FUNCTION_BLOCK PalletizerConveyor EXTENDS Conveyor
VAR_INPUT
END_VAR
VAR_OUTPUT
	bStartBackward : BOOL;
END_VAR
VAR	
	fbStartBackward : BoolOut;
END_VAR

SUPER^();
bStartBackward := fbStartBackward.getValue;

PROPERTY getStartBackward : BoolOut
GET
getStartBackward := fbStartBackward;
END_GET
END_PROPERTY

END_FUNCTION_BLOCK

(* stored: Version 1.1.0.1, ProductVersion 3.1.4024.0
   POU PalletizerConveyor: Id {fedbe3e3-7fa7-4ce9-a006-c2d0089d037d}, SpecialFunc None
   Property getStartBackward: Id {117b1f55-dc43-4a43-93cf-132871f6c536}
   Get Get: Id {a41fe51c-870b-4bfe-be0f-d61351090d79} *)
